{attribute addProperty BoxType "EJ7211-0011-0026"}
{attribute addProperty Id "ControlwordAT %Q*UINT162"}
{attribute addProperty CRC "1098258280"}
{attribute addProperty SizeInBites "16"}
{attribute addProperty SizeInBytes "2"}
TYPE DS402_Controlword_41761768 :
STRUCT
	{attribute addProperty Name "Controlword"}
	Controlword AT %Q* : UINT;
END_STRUCT
END_TYPE

(* stored: Version 1.2.0.0, ProductVersion 3.1.4024.9
   DUT DS402_Controlword_41761768: Id {1b75f584-6ce8-4e16-a28a-3485a2a4e0a5} *)
